PROGRAM Outputs_RB
VAR
	HmiPBDoorRequest: BOOL;
	HmiPBIndexFwd: BOOL;
	HmiPBIndexRev: BOOL;
	HmiPBDustCollect: BOOL;
	HmiPBSawStart: BOOL;
	HmiPBSawStop: BOOL;
	HmiPBTraverseFwd: BOOL;
	HmiPBTraverseRev: BOOL;
	HmiPBLiftRaise: BOOL;
	HmiPBLiftLower: BOOL;
	HmiPBTransferFwd: BOOL;
	HmiPBTransferRev: BOOL;
	HmiPBTransferClampOpen: BOOL;
	HmiPBTransferClampClose: BOOL;
	HmiPBTransferClampFwd: BOOL;
	HmiPBTransferClampRev: BOOL;
	HmiPBSawClampClose: BOOL;
	HmiPBSawClampOpen: BOOL;
	HmiPBSawClampFwd: BOOL;
	HmiPBSawClampRev: BOOL;
	HmiPBPinsRaise: BOOL;
	HmiPBPinsLower: BOOL;
	
	
	
	
END_VAR

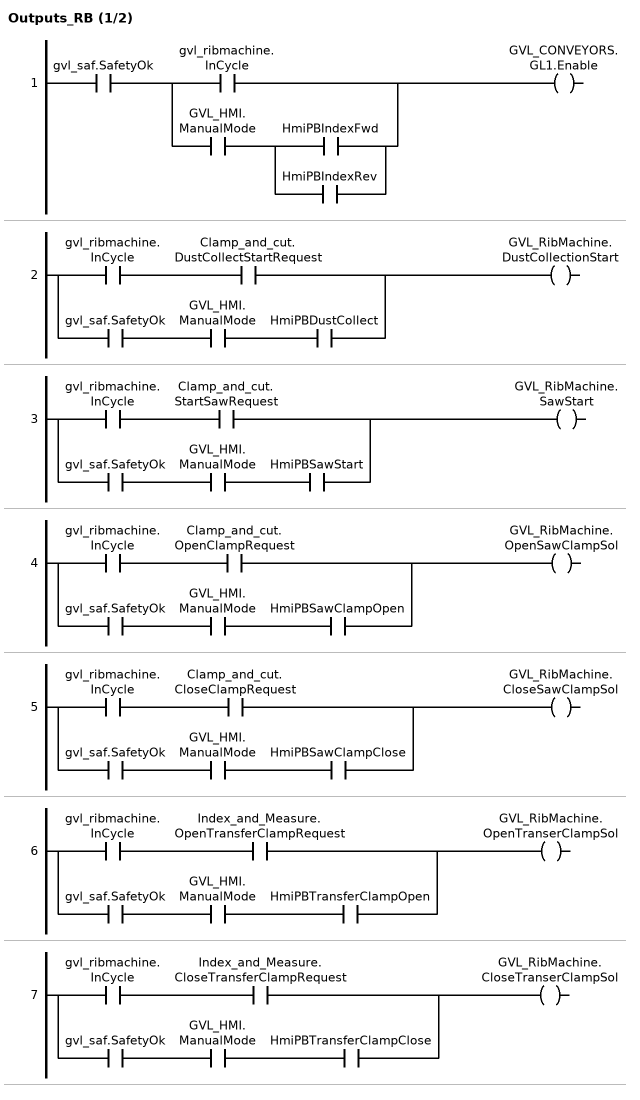
// NETWORK 1
GVL_CONVEYORS.GL1.Enable := gvl_saf.SafetyOk AND (gvl_ribmachine.InCycle OR GVL_HMI.ManualMode AND (HmiPBIndexFwd OR HmiPBIndexRev));

// NETWORK 2
GVL_RibMachine.DustCollectionStart := gvl_ribmachine.InCycle AND Clamp_and_cut.DustCollectStartRequest OR gvl_saf.SafetyOk AND GVL_HMI.ManualMode AND HmiPBDustCollect;

// NETWORK 3
GVL_RibMachine.SawStart := gvl_ribmachine.InCycle AND Clamp_and_cut.StartSawRequest OR gvl_saf.SafetyOk AND GVL_HMI.ManualMode AND HmiPBSawStart;

// NETWORK 4
GVL_RibMachine.OpenSawClampSol := gvl_ribmachine.InCycle AND Clamp_and_cut.OpenClampRequest OR gvl_saf.SafetyOk AND GVL_HMI.ManualMode AND HmiPBSawClampOpen;

// NETWORK 5
GVL_RibMachine.CloseSawClampSol := gvl_ribmachine.InCycle AND Clamp_and_cut.CloseClampRequest OR gvl_saf.SafetyOk AND GVL_HMI.ManualMode AND HmiPBSawClampClose;

// NETWORK 6
GVL_RibMachine.OpenTranserClampSol := gvl_ribmachine.InCycle AND Index_and_Measure.OpenTransferClampRequest OR gvl_saf.SafetyOk AND GVL_HMI.ManualMode AND HmiPBTransferClampOpen;

// NETWORK 7
GVL_RibMachine.CloseTranserClampSol := gvl_ribmachine.InCycle AND Index_and_Measure.CloseTransferClampRequest OR gvl_saf.SafetyOk AND GVL_HMI.ManualMode AND HmiPBTransferClampClose;

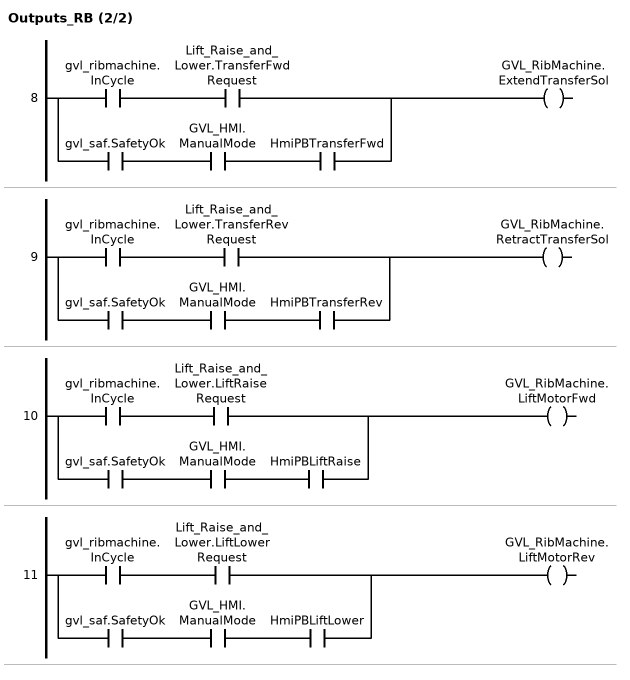
// NETWORK 8
GVL_RibMachine.ExtendTransferSol := gvl_ribmachine.InCycle AND Lift_Raise_and_Lower.TransferFwdRequest OR gvl_saf.SafetyOk AND GVL_HMI.ManualMode AND HmiPBTransferFwd;

// NETWORK 9
GVL_RibMachine.RetractTransferSol := gvl_ribmachine.InCycle AND Lift_Raise_and_Lower.TransferRevRequest OR gvl_saf.SafetyOk AND GVL_HMI.ManualMode AND HmiPBTransferRev;

// NETWORK 10
GVL_RibMachine.LiftMotorFwd := gvl_ribmachine.InCycle AND Lift_Raise_and_Lower.LiftRaiseRequest OR gvl_saf.SafetyOk AND GVL_HMI.ManualMode AND HmiPBLiftRaise;

// NETWORK 11
GVL_RibMachine.LiftMotorRev := gvl_ribmachine.InCycle AND Lift_Raise_and_Lower.LiftLowerRequest OR gvl_saf.SafetyOk AND GVL_HMI.ManualMode AND HmiPBLiftLower;

END_PROGRAM

(* stored: Version 1.1.0.1, ProductVersion 3.1.4024.12
   POU Outputs_RB: Id {5e3b8410-f955-4f9e-b751-30e3dad9c258}, SpecialFunc None *)
